# B&R Automation Studio project MiguelA214Projeto
Automation Studio 4.1.14.40 SP

## Configuration Config1

CPU X20CP1583, AutomationRuntime D4.09, Build 4.1.2, Vc V4.15.9

### Task classes (Cpu.sw)
```
Cyclic#4 (cycle 100000 us, tolerance 100000 us):
  ProjetoMig <- ProjetoMiguelA214.prg
Libraries: standard
```

### Hardware
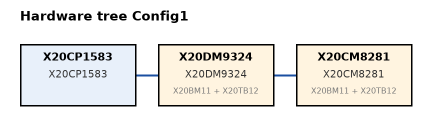
```
X20BM11 : X20BM11 v1.0.0.0  [X2X1 -> X20CP1583.IF6]
X20BM11a : X20BM11 v1.0.0.0  [X2X1 -> X20BM11.X2X2]
X20CM8281 : X20CM8281 v1.0.3.0  [SS1 -> X20TB12a.SS; SL -> X20BM11a.SL1]
X20CP1583 : X20CP1583 v1.0.4.0
  Connector IF2:
    ActivateDevice = 1
    EthInterfaceRedundant = 0
    Mode = Manual
    InternetAddress = 192.168.0.70
    SubnetMask = 255.255.255.0
  Connector IF3:
    EplInterfaceRedundant = 0
    EplEthInterfaceRedundant = 0
  ConfigurationID = MiguelA214Projeto_Config1
  TimerDeviceType = SWIOTIMER
  Cyclic1Duration = 10000
  Cyclic1Tolerance = 10000
  Cyclic2Duration = 20000
  Cyclic2Tolerance = 20000
  Cyclic3Duration = 50000
  Cyclic3Tolerance = 50000
  Cyclic4Duration = 100000
  Cyclic4Tolerance = 100000
  Cyclic5Duration = 200000
  Cyclic5Tolerance = 200000
  Cyclic6Duration = 500000
  Cyclic6Tolerance = 500000
  Cyclic7Duration = 1000000
  Cyclic7Tolerance = 1000000
  Cyclic8Duration = 10000
  Cyclic8Tolerance = 30000000
  ActivateOpcUa = 1
  OpcUaAnonymous = 1
  OpcUaAnonymousAccess = 1
X20DM9324 : X20DM9324 v1.0.1.0  [SS1 -> X20TB12.SS; SL -> X20BM11.SL1]
X20TB12 : X20TB12 v1.0.0.0
X20TB12a : X20TB12 v1.0.0.0
```

### IoMap.iom - X20CP1583/IoMap.iom
```iecst
(********************************************************************
 * COPYRIGHT --
 ********************************************************************
 * File: IoMap.iom
 * Author: supervisorio
 * Created: June 12, 2024
 ********************************************************************
 * IO mapping file
 ********************************************************************)
VAR_CONFIG
	::ProjetoMig:BIT1 AT %QX."X20CM8281".DigitalOutput01;
	::ProjetoMig:BIT0 AT %QX."X20CM8281".DigitalOutput02;
	::ProjetoMig:BIT5 AT %QX."X20DM9324".DigitalOutput01;
	::ProjetoMig:BIT4 AT %QX."X20DM9324".DigitalOutput02;
	::ProjetoMig:BIT3 AT %QX."X20DM9324".DigitalOutput03;
	::ProjetoMig:BIT2 AT %QX."X20DM9324".DigitalOutput04;
END_VAR
```

## Logical view

Binary libraries used (declarations not repeated): operator, runtime, astime, AsIecCon, standard

### Global.var - Global variables
```iecst
VAR
	ORIGEM : INT;
	DESTINO : INT;
	START_MOVE : BOOL;
END_VAR
```


### Program Logical/ProjetoMiguelA214 (IEC) - Program

#### ProjetoMiguelA214Cyclic.st - Cyclic code
```iecst
(********************************************************************
 * COPYRIGHT --
 ********************************************************************
 * Program: ProjetoMiguelA214
 * File: ProjetoMiguelA214Cyclic.st
 * Author: supervisorio
 * Created: June 12, 2024
 ********************************************************************
 * Implementation of program ProjetoMiguelA214
 ********************************************************************)

PROGRAM _CYCLIC

	IF EDGEPOS(START_MOVE) THEN
		IF (0 < ORIGEM) AND (ORIGEM <= 12) AND (0 < DESTINO) AND (DESTINO <= 12) THEN
			SAIDA := ORIGEM - 1; (*Define origem*)
			TI.IN := TRUE;
		ELSE
			START_MOVE := FALSE;
		END_IF;
	END_IF;

	IF TI.Q THEN
		TI.IN := FALSE;
		TI2.IN := TRUE;
		SAIDA := SAIDA + 16; (*Muda o 5º bit primeiro pra garantir que a origem não modifique*)
	END_IF;

	IF TI2.Q THEN
		TI2.IN := FALSE;
		TI3.IN := TRUE;
		SAIDA := DESTINO + 16 - 1; (*Define destino*)
	END_IF;

	IF TI3.Q THEN
		TI3.IN := FALSE;
		TI4.IN := TRUE;
		SAIDA := SAIDA + 32; (*Inicia movimentação*)
	END_IF;

	IF TI4.Q THEN
		TI4.IN := FALSE;
		START_MOVE := FALSE;
		SAIDA := 0;
	END_IF;

	BIT0 := SAIDA.0;
	BIT1 := SAIDA.1;
	BIT2 := SAIDA.2;
	BIT3 := SAIDA.3;
	BIT4 := SAIDA.4;
	BIT5 := SAIDA.5;

	TI.PT := T#100ms;
	TI();
	TI2.PT := T#100ms;
	TI2();
	TI3.PT := T#100ms;
	TI3();
	TI4.PT := T#100ms;
	TI4();

END_PROGRAM
```

#### ProjetoMiguelA214.var - Local variables
```iecst
(********************************************************************
 * COPYRIGHT --
 ********************************************************************
 * Program: ProjetoMiguelA214
 * File: ProjetoMiguelA214.var
 * Author: supervisorio
 * Created: June 12, 2024
 ********************************************************************
 * Local variables of program ProjetoMiguelA214
 ********************************************************************)
VAR
	SAIDA : INT;
	TI : TON;
	TI2 : TON;
	TI3 : TON;
	BIT0 : BOOL;
	BIT1 : BOOL;
	BIT2 : BOOL;
	BIT3 : BOOL;
	BIT4 : BOOL;
	BIT5 : BOOL;
	TI4 : TON;
END_VAR
```
